{attribute addProperty BoxType "EL5072-0000-0016"}
{attribute addProperty Id "IND_Inputs_ChannelAT %I*ARRAY[0..1] OF IND_Inputs_Channel_F11037BF160200IND_Outputs_ChannelAT %Q*ARRAY[0..1] OF IND_Outputs_Channel_CDB9543D112140WcStateAT %I*WcState_F855686C1620InfoDataAT %I*InfoData_BC63D37F80100"}
{attribute addProperty CRC "3341612877"}
{attribute addProperty SizeInBites "368"}
{attribute addProperty SizeInBytes "46"}
TYPE EL5072_B22199CB :
STRUCT
	{attribute addProperty Name "IND_Inputs_Channel"}
	IND_Inputs_Channel : ARRAY[0..1] OF IND_Inputs_Channel_F11037BF;
	{attribute addProperty Name "IND_Outputs_Channel"}
	IND_Outputs_Channel : ARRAY[0..1] OF IND_Outputs_Channel_CDB9543D;
	{attribute addProperty Name "WcState"}
	WcState : WcState_F855686C;
	{attribute addProperty Name "InfoData"}
	InfoData : InfoData_BC63D37F;
END_STRUCT
END_TYPE

(* stored: Version 1.2.0.0, ProductVersion 3.1.4024.9
   DUT EL5072_B22199CB: Id {6ac373c7-c99c-4afd-92fa-eb3227c98f48} *)
